FUNCTION_BLOCK L0_CompletedEx (* Basic Function Block Type *)
  (* Standard: 61499-2 *)
  (* Version 0.0, 2014-09-04, EQUEROL, UJI *)
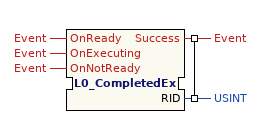
  EVENT_INPUT
    OnReady; (* CNC Ready event *)
    OnExecuting; (* CNC Executing event *)
    OnNotReady; (* CNC NotReadyEvent *)
  END_EVENT
  EVENT_OUTPUT
    Success WITH RID; (* Execution succed *)
  END_EVENT
  VAR_OUTPUT
    RID : USINT; (* Execution returned ID *)
  END_VAR
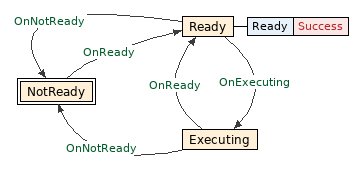
  EC_STATES
    NotReady; (* Initial State *)
    Ready : Ready -> Success; (* Initialization *)
    Executing; (* Normal execution *)
  END_STATES
  EC_TRANSITIONS
    NotReady TO Ready := OnReady;
    Ready TO Executing := OnExecuting;
    Executing TO Ready := OnReady;
    Executing TO NotReady := OnNotReady;
    Ready TO NotReady := OnNotReady;
  END_TRANSITIONS
  ALGORITHM Ready IN ST: (* Successful action algo *)
RID:=0;
  END_ALGORITHM
END_FUNCTION_BLOCK
